// Mitsubishi GX Works2 project: 5   PLC: FX2N/FX2NC

PROGRAM MAIN
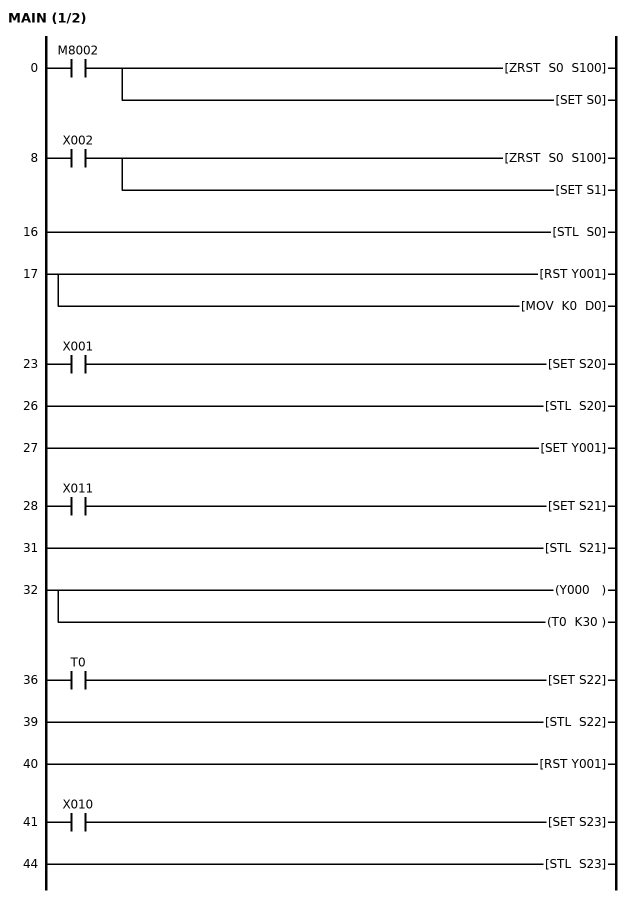
0     LD      M8002
      ZRST    S0 S100
      SET     S0
8     LD      X002
      ZRST    S0 S100
      SET     S1
16    STL     S0
17    RST     Y001
      MOV     K0 D0
23    LD      X001
      SET     S20
26    STL     S20
27    SET     Y001
28    LD      X011
      SET     S21
31    STL     S21
32    OUT     Y000
      OUT     T0 K30
36    LD      T0
      SET     S22
39    STL     S22
40    RST     Y001
41    LD      X010
      SET     S23
44    STL     S23
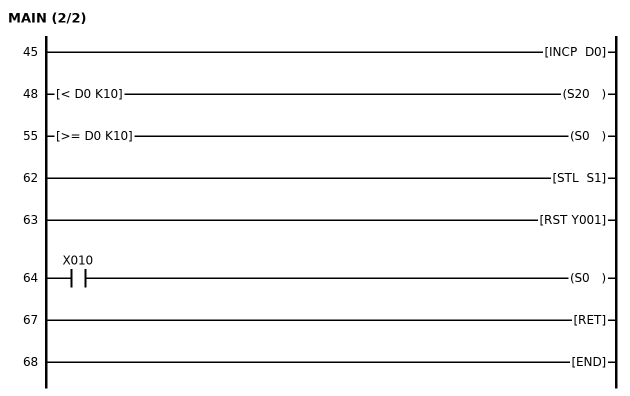
45    INCP    D0
48    LD<     D0 K10
      OUT     S20
55    LD>=    D0 K10
      OUT     S0
62    STL     S1
63    RST     Y001
64    LD      X010
      OUT     S0
67    RET
68    END
END_PROGRAM

// device comments not shown above
BL0  ; main
BL1  ; a
BL2  ; b
